(* CODESYS project DigitalInput_0.0.2.library
   Description: Function Block designed to interface with digital inputs for easy programming.
   Version: 0.0.2
   Title: DigitalInput
   Author: Ali Alam
   Placeholder: DigitalInput
   Company: Promise Robotics

Project tree, tasks and I/O mapping:
  libraries: Tc2_Standard, * (Beckhoff Automation GmbH); Tc2_System, * (Beckhoff Automation GmbH)
  DUTs/
  GVLs/
  POUs/
    function block FB_DigitalInput [ST]: P_DebounceTime, P_Value
    interface ITF_DigitalInput: P_DebounceTime, P_Value
  VISUs/
*)

// POUs/FB_DigitalInput
FUNCTION_BLOCK FB_DigitalInput IMPLEMENTS ITF_DigitalInput
VAR_INPUT
	{ attribute 'TcHmiSymbol.AddSymbol' }
	RawInput AT %I*   : BOOL;
END_VAR
VAR
	{ attribute 'TcHmiSymbol.AddSymbol' }
	DebounceTime      : TIME := T#0MS;
	DebounceTimer     : TON;
	
	PrevState		  : BOOL := FALSE;
	{ attribute 'TcHmiSymbol.AddSymbol' }
	Value		  	  : BOOL := FALSE;
END_VAR

PROPERTY P_DebounceTime : TIME
SET
DebounceTime := P_DebounceTime;
END_SET
END_PROPERTY

PROPERTY P_Value : BOOL
GET
IF DebounceTime = T#0MS THEN // No Debounce set
	P_Value := RawInput; 
ELSE                         // Debounce set
	IF RawInput <> PrevState THEN
    	DebounceTimer(IN := TRUE, PT := DebounceTime);
	ELSE
		DebounceTimer(IN := FALSE);
	END_IF
	
	// When debounce time has passed and input is stable
	IF DebounceTimer.Q THEN
		Value := RawInput;
		PrevState := RawInput;
	END_IF
	
	P_Value := Value;
END_IF
END_GET
END_PROPERTY

END_FUNCTION_BLOCK

// POUs/ITF_DigitalInput
INTERFACE ITF_DigitalInput

PROPERTY P_DebounceTime : TIME
SET
END_SET
END_PROPERTY

PROPERTY P_Value : BOOL
GET
END_GET
END_PROPERTY

END_INTERFACE
